TYPE ST_PersistentData_02 :
STRUCT
	nData01		: DINT;
	nData02		: INT;
	fData03		: LREAL;
	bTest01		: BOOL;
	nTest02		: INT;
END_STRUCT
END_TYPE

(* stored: Version 1.1.0.1, ProductVersion 3.1.4024.6
   DUT ST_PersistentData_02: Id {e691dc8f-131d-476c-a4ba-055d5b02d270} *)
